// Mitsubishi GX Developer project: HOME_CONTROLLER_FX3U   PLC: FX3U

PROGRAM MAIN
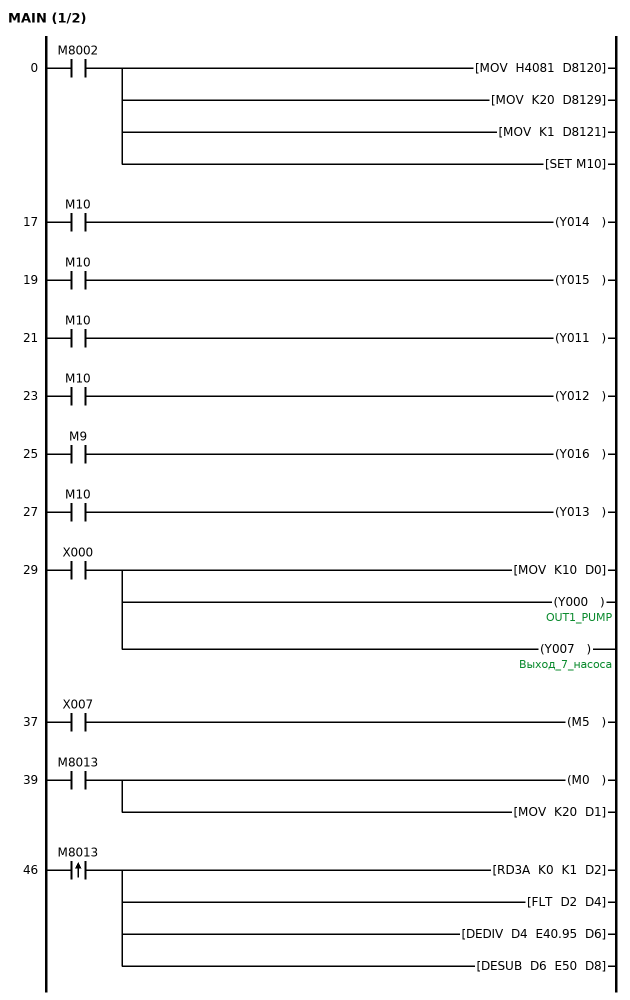
0     LD      M8002
      MOV     H4081 D8120
      MOV     K20 D8129
      MOV     K1 D8121
      SET     M10
17    LD      M10
      OUT     Y014
19    LD      M10
      OUT     Y015
21    LD      M10
      OUT     Y011
23    LD      M10
      OUT     Y012
        [note] Y14
25    LD      M9
      OUT     Y016
27    LD      M10
      OUT     Y013
29    LD      X000
      MOV     K10 D0
        [note] Discret output (coil) -t 0
      OUT     Y000  ; OUT1_PUMP
        [note] -t 1 [257][4353]
      OUT     Y007  ; Выход_7_насоса
        [note] -t1 [264] [4360]
37    LD      X007
      OUT     M5
39    LD      M8013
      OUT     M0
      MOV     K20 D1
46    LDP     M8013
      RD3A    K0 K1 D2
      FLT     D2 D4
      DEDIV   D4 E40.95 D6
      DESUB   D6 E50 D8
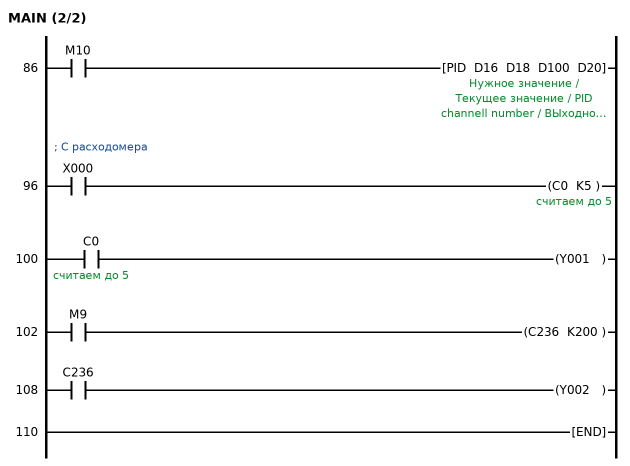
86    LD      M10
      PID     D16 D18 D100 D20  ; Нужное значение / Текущее значение / PID channell number / ВЫходное значение
; С расходомера
96    LD      X000
      OUT     C0 K5  ; считаем до 5
        [note] Будем считать
100   LD      C0  ; считаем до 5
      OUT     Y001
102   LD      M9
      OUT     C236 K200
108   LD      C236
      OUT     Y002
110   END
END_PROGRAM

// device comments not shown above
D101  ; PID ratior koeff KP
D102  ; PID KI
D103  ; PID KD
D104  ; PID KE (error)
D105  ; PID PMAX
D106  ; PID PMIN
D107  ; PID backup
D108  ; PID standbay
